FUNCTION F_LWORD_ARG : ST_Arg
VAR_INPUT
	lwInput : LWORD;
END_VAR
VAR
	stArg : ST_Arg;
	sysVar_Info : __SYSTEM.VAR_INFO;
END_VAR

sysVar_Info 	:= __VARINFO(lwInput);
stArg.TypeClass := sysVar_Info.TypeClass;
stArg.pValue 	:= 0;
stArg.diSize 	:= SIZEOF(lwInput);
stArg.sValue 	:= TO_STRING(lwInput); 
F_LWORD_ARG := stArg;

END_FUNCTION

(* stored: Version 1.1.0.1, ProductVersion 3.1.4024.4
   POU F_LWORD_ARG: Id {a0b4b68e-62c0-4492-ace0-880a7173624c}, SpecialFunc None *)
